PROGRAM ComplexExercises

END_PROGRAM

(* stored: Version 1.1.0.1
   POU ComplexExercises: Id {d3591d61-8c3a-4082-b225-3ff7b75cc993}, SpecialFunc None *)
